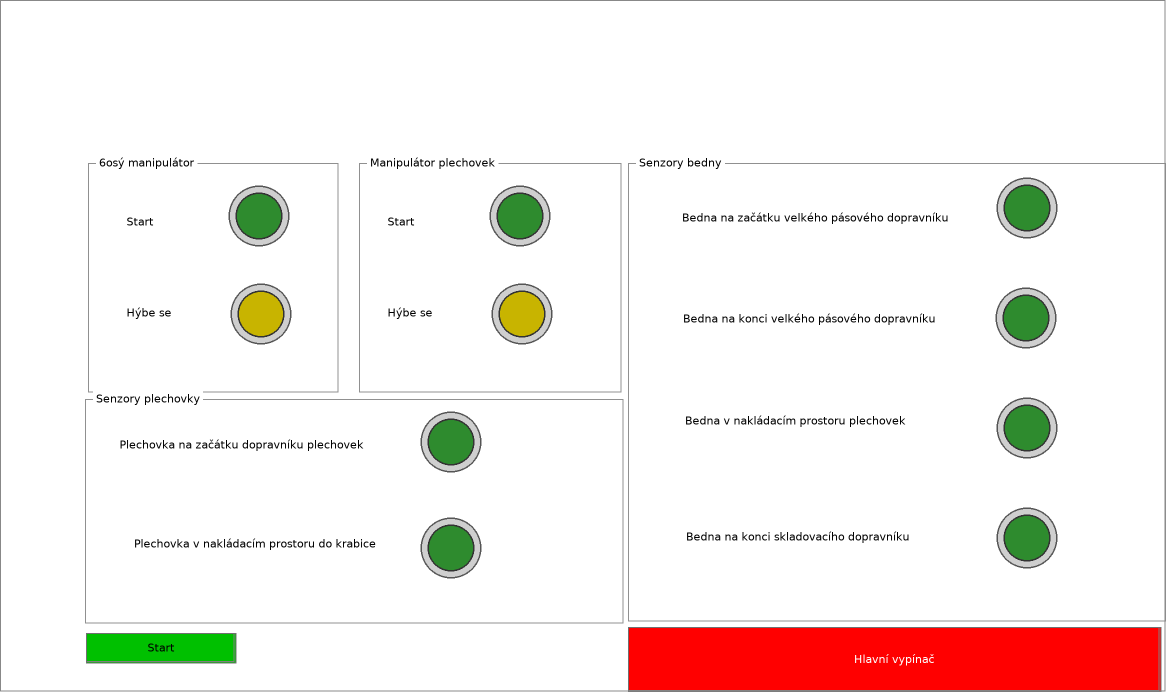
VISUALIZATION Visualization  // 1166x692
    Lamp1 (992,173 70x70), variable: IO.SensorBoxStart, style: Lamp-Lamp1-Green
    Lamp1 (991,283 70x70), variable: IO.SensorBoxHandled, style: Lamp-Lamp1-Green
    Label (669,203 293x30), "Bedna na začátku velkého pásového dopravníku"
    Label (663,304 293x30), "Bedna na konci velkého pásového dopravníku"
    Lamp1 (992,393 70x70), variable: IO.SensorBoxHandling, style: Lamp-Lamp1-Green
    Label (644,406 303x30), "Bedna v nakládacím prostoru plechovek"
    Lamp1 (992,503 70x70), variable: IO.SensorBoxStoring, style: Lamp-Lamp1-Green
    Label (668,522 260x30), "Bedna na konci skladovacího dopravníku"
    GroupBox (628,155 538x466), "Senzory bedny"
    Lamp1 (485,181 70x70), variable: IO.HandlingStartCycle, style: Lamp-Lamp1-Green
    Label (356,301 108x24), "Hýbe se"
    Lamp1 (487,279 70x70), variable: IO.HandlingMoving, style: Lamp-Lamp1-Yellow
    Label (347,208 108x28), "Start"
    Lamp1 (224,181 70x70), variable: IO.RoboticArmStartCycle, style: Lamp-Lamp1-Green
    Label (95,301 108x24), "Hýbe se"
    Lamp1 (226,279 70x70), variable: IO.RoboticArmMoving, style: Lamp-Lamp1-Yellow
    Label (86,208 108x28), "Start"
    GroupBox (88,155 250x237), "6osý manipulátor"
    GroupBox (359,155 262x237), "Manipulátor plechovek"
    Button (628,627 533x65), "Hlavní vypínač", invisible if: MAIN.StartProcess
        toggle MAIN.CentralStop
    Button (86,633 150x30), "Start"
        toggle MAIN.StartProcess
    Lamp1 (416,407 70x70), variable: IO.SensorCanNew, style: Lamp-Lamp1-Green
    Label (114,430 255x30), "Plechovka na začátku dopravníku plechovek"
    Lamp1 (416,513 70x70), variable: IO.SensorCanHandling, style: Lamp-Lamp1-Green
    GroupBox (85,391 538x232), "Senzory plechovky"
    Label (118,529 274x30), "Plechovka v nakládacím prostoru do krabice"
END_VISUALIZATION

(* stored: Version 1.1.0.1, ProductVersion 3.1.4024.15
   Visu Visualization: Id {6aba3b2b-f4f4-47a7-8832-28cd1880003e} *)
